FUNCTION_BLOCK FB_RollRightAngle
VAR_INPUT
	ref_Roller 	:REFERENCE TO ST_Inventer;
	ref_Belt 	:REFERENCE TO ST_Inventer;
	ref_UD 		:REFERENCE TO ST_InventerUD;
END_VAR
VAR_OUTPUT
	o_bError :BOOL;
END_VAR
VAR
	_Belt	:BOOL;
	ldfBeltOff	:F_TRIG;
	
	_Roller	:BOOL;
	tmrRollerDelay	:TON;
	ldfRollerOff	:F_TRIG;
	
	tmrErrorDelay	:TON;
END_VAR

//Error cont.
o_bError := ref_Belt.iError	OR ref_Roller.iError OR ref_UD.iError OR  tmrErrorDelay.Q;





//皮帶
ldfBeltOff(CLK:=_Belt);
IF ldfBeltOff.q THEN
	tmrErrorDelay(IN:=FALSE);
	ref_Belt.qRun	:=FALSE;
	ref_UD.qSign	:= FALSE;
	ref_UD.qRun		:= FALSE;
END_IF
_Belt	:=FALSE;


//進入滾珠
ldfRollerOff(CLK:=_Roller);

IF ldfRollerOff.Q THEN
	tmrErrorDelay(IN:=FALSE);
	tmrRollerDelay(IN:=FALSE);
	ref_Roller.qRun	:=FALSE;
	ref_UD.qSign	:= FALSE;
	ref_UD.qRun		:= FALSE;
END_IF

_Roller	:=FALSE;

METHOD Belt : BOOL
VAR_INPUT
END_VAR
_Belt	:= TRUE;
ref_Belt.qRun	:= TRUE;
//Error Timer 
tmrErrorDelay(IN:=NOT ref_UD.iHighPos,PT:=T#2S);
//belt In senser Position 
ref_UD.qRun	:= NOT ref_UD.iHighPos;
ref_UD.qSign		:= FALSE;


IF tmrErrorDelay.Q THEN
	ref_UD.qSign	:= FALSE;
	ref_UD.qRun		:= FALSE;
END_IF
END_METHOD

METHOD Initialization : BOOL
VAR_INPUT
END_VAR
_Roller	:= TRUE;
ref_Roller.qRun	:= FALSE;
ref_Belt.qRun	:= FALSE;
//Error Timer 
tmrErrorDelay(IN:=NOT ref_UD.iLowPos,PT:=T#2S);
//
IF NOT ref_UD.iLowPos THEN
	ref_UD.qSign	:= TRUE;
	tmrRollerDelay(IN:=TRUE,PT:= T#20MS);
	ref_UD.qRun	:= tmrRollerDelay.Q ;
	ELSE
	ref_UD.qSign	:= FALSE;
	ref_UD.qRun		:= FALSE;
END_IF

Initialization	:= ref_UD.iLowPos;
END_METHOD

METHOD Roller : BOOL
VAR_INPUT
END_VAR
_Roller	:= TRUE;
ref_Belt.qRun	:= FALSE;
//Error Timer 
tmrErrorDelay(IN:=NOT ref_UD.iLowPos,PT:=T#2S);
//
IF NOT ref_UD.iLowPos THEN
	ref_UD.qSign	:= TRUE;
	tmrRollerDelay(IN:=TRUE,PT:= T#20MS);
	ref_UD.qRun	:= tmrRollerDelay.Q ;
	ELSE
	ref_UD.qSign	:= FALSE;
	ref_UD.qRun		:= FALSE;
	ref_Roller.qRun	:= TRUE	;
END_IF


IF tmrErrorDelay.Q THEN
	ref_UD.qSign	:= FALSE;
	ref_UD.qRun		:= FALSE;
END_IF
END_METHOD

END_FUNCTION_BLOCK

(* stored: Version 1.1.0.1, ProductVersion 3.1.4024.16
   POU FB_RollRightAngle: Id {368a9ff0-37f2-4291-a208-b58d431d0df0}, SpecialFunc None
   Method Belt: Id {c3238a18-d7f1-4acd-81a9-eb2d65650f73}
   Method Initialization: Id {0220c0b0-f9db-4911-a89c-5db7995b6a52}
   Method Roller: Id {04ee8195-5588-4573-8357-a2e371727927} *)
